{attribute 'qualified_only'}
{attribute 'strict'}
{attribute 'to_string'}
TYPE E_BaseEvents_Type :
(
	BRAK		:= 0,
	BLAD		:= 1, 
	ALARM		:= 2, 
	SAFETY		:= 3, 
	WIADOMOSC	:= 4

);
END_TYPE

(* stored: Version 1.1.0.1
   DUT E_BaseEvents_Type: Id {aee22ca8-38f0-4d5e-8215-120a4a034c27} *)
